{attribute addProperty BoxType "EPP1342-0001-0016"}
{attribute addProperty Id "A_0024_EPP1342_0001_0017A_0024_EPP1342_0001_0017_B861A0082662332.75"}
{attribute addProperty CRC "4079902448"}
{attribute addProperty SizeInBites "2662"}
{attribute addProperty SizeInBytes "332.75"}
TYPE A_0023_EPP1342_0001_0016_F32E5EF0 EXTENDS EPP1342_179A0949 :
STRUCT
	{attribute addProperty Name "A_0024_EPP1342_0001_0017"}
	A_0024_EPP1342_0001_0017 : A_0024_EPP1342_0001_0017_B861A008;
END_STRUCT
END_TYPE

(* stored: Version 1.2.0.0, ProductVersion 3.1.4024.9
   DUT A_0023_EPP1342_0001_0016_F32E5EF0: Id {ad90f48e-659e-4253-9abc-f12eb28cddb3} *)
